TYPE stBH0GPL_Line EXTENDS stPIM_LineEventsModule :
STRUCT

	{attribute 'OPC.UA.DA' := '1'}
	stStation_BH0GPL01 : stPIM_StationEventsModule_3_Machine;
END_STRUCT
END_TYPE

(* stored: Version 1.1.0.1, ProductVersion 3.1.4024.15
   DUT stBH0GPL_Line: Id {f2493a5d-fb56-447f-9fe1-2792dc7570a7} *)
